{attribute addProperty BoxType "EL6201-0000-0017"}
{attribute addProperty Id "Auto_Programming_EnableAT %Q*BOOL811Go_Offline_ModeAT %Q*BOOL812Data_Exchange_ActiveAT %Q*BOOL813Go_Protected_ModeAT %Q*BOOL814Go_Configuration_ModeAT %Q*BOOL815"}
{attribute addProperty CRC "1016930845"}
{attribute addProperty SizeInBites "40"}
{attribute addProperty SizeInBytes "5"}
TYPE ASI_Control_3C9D221D :
STRUCT
	{attribute addProperty Name "Auto_Programming_Enable"}
	Auto_Programming_Enable AT %Q* : BOOL;
	{attribute addProperty Name "Go_Offline_Mode"}
	Go_Offline_Mode AT %Q* : BOOL;
	{attribute addProperty Name "Data_Exchange_Active"}
	Data_Exchange_Active AT %Q* : BOOL;
	{attribute addProperty Name "Go_Protected_Mode"}
	Go_Protected_Mode AT %Q* : BOOL;
	{attribute addProperty Name "Go_Configuration_Mode"}
	Go_Configuration_Mode AT %Q* : BOOL;
END_STRUCT
END_TYPE

(* stored: Version 1.2.0.0, ProductVersion 3.1.4024.9
   DUT ASI_Control_3C9D221D: Id {943bae1f-cf37-4068-aed8-fd8e50d1269e} *)
